Fanuc KAREL source: ka00121.KL

-- PROVISIONAL review KL for V770-1; original PC SHA256 c52ee7a00ea0683a54c6c68b8169e1aa1424cd8510b25eba75b4708a7cf9c492
-- Incomplete behavior may be omitted. Consult companion uncertainty JSON. Do not deploy.
PROGRAM KA00121
%NOLOCKGROUP
VAR
  DST : INTEGER
-- UNRESOLVED_DECL SRC type=002018
BEGIN
  -- UNRESOLVED_PC offsets 5-19; opcodes 2E,22,9D,33,B2
  -- UNRESOLVED_PC offsets 24-39; opcodes 22,9D,33,B1,23
  -- UNRESOLVED_PC offsets 44-48; opcodes 7F
END KA00121
